{attribute 'qualified_only'}
VAR_GLOBAL
	
(*Variables for the first DI-card*)
	di01 AT %IX0.0 : BOOL;
	di02 AT %IX0.1 : BOOL;
	di03 AT %IX0.2 : BOOL;
	di04 AT %IX0.3 : BOOL;
	di05 AT %IX0.4 : BOOL;
	di06 AT %IX0.5 : BOOL;
	di07 AT %IX0.6 : BOOL;
	di08 AT %IX0.7 : BOOL;
	
END_VAR

(* stored: Version 1.1.0.1, ProductVersion 3.1.4020.12
   GVL IOlinks: Id {16c8edf1-c74c-4f53-a50e-07c773513886} *)
